// TwinCAT 3 PLC project Untitled1
// ProgramVersion: 3.1.4024.0
// libraries:
//   Tc2_Standard, * (Beckhoff Automation GmbH)
//   Tc2_System, * (Beckhoff Automation GmbH)
//   Tc3_Module, * (Beckhoff Automation GmbH)
// project tree:
//   / PlcTask.TcTTO
//   POUs/ MAIN.TcPOU

CONFIGURATION Untitled1
    RESOURCE PLC ON TwinCAT3
        TASK PlcTask(INTERVAL := T#10ms, PRIORITY := 21);
        PROGRAM MAIN WITH PlcTask : MAIN;
    END_RESOURCE
END_CONFIGURATION

// ---- POUs/MAIN.TcPOU
PROGRAM MAIN
VAR
status: INT;
Vision: BOOL;
Trig AT %Q*: BOOL;
Out AT %I*: BOOL;
Button AT %I*: BOOL;
pick: BOOL;
reset AT %I*: BOOL;
//request AT %I*: BOOL;
END_VAR;

CASE status OF
	
0: 	IF Button = TRUE THEN
	Trig := TRUE;
	ELSE Trig := FALSE;
	END_IF
	
	IF Out = TRUE THEN	
		status := 1;
	END_IF
	
	IF reset = TRUE THEN
		pick := FALSE;
	END_IF
	
1: IF Button = TRUE THEN
	Trig := TRUE;
	ELSE Trig := FALSE;
	END_IF
	
	IF Out = FALSE THEN	
		pick := TRUE;
		status := 0;	
	END_IF
	
	IF reset = TRUE THEN
		pick := FALSE;
	END_IF
	
END_CASE

END_PROGRAM
